PROGRAM PRG_91_TwinSAFE
VAR
	FB_Blinker_Estop: FB_Blinker;
END_VAR
VAR // added by the converter: edge detectors and wires of the graphical bodies
    _w1, _w2, _w3 : BOOL;
END_VAR

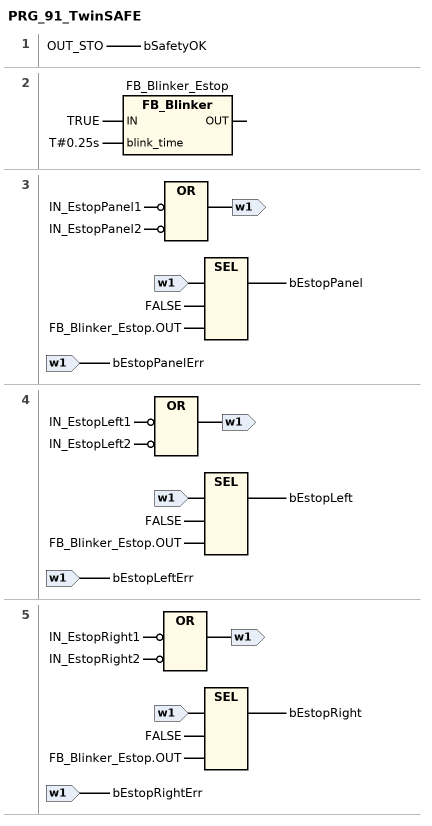
// NETWORK 1
bSafetyOK := OUT_STO;

// NETWORK 2
FB_Blinker_Estop(IN := TRUE, blink_time := T#0.25s); // FB_Blinker

// NETWORK 3
_w1 := NOT IN_EstopPanel1 OR NOT IN_EstopPanel2;
bEstopPanel := SEL(_w1, FALSE, FB_Blinker_Estop.OUT);
bEstopPanelErr := _w1;

// NETWORK 4
_w2 := NOT IN_EstopLeft1 OR NOT IN_EstopLeft2;
bEstopLeft := SEL(_w2, FALSE, FB_Blinker_Estop.OUT);
bEstopLeftErr := _w2;

// NETWORK 5
_w3 := NOT IN_EstopRight1 OR NOT IN_EstopRight2;
bEstopRight := SEL(_w3, FALSE, FB_Blinker_Estop.OUT);
bEstopRightErr := _w3;

END_PROGRAM

(* stored: Version 1.1.0.1, ProductVersion 3.1.4024.15
   POU PRG_91_TwinSAFE: Id {b6afbb74-a48b-4472-b228-a2fe61b4c86d}, SpecialFunc None *)
